PROGRAM TELNET_PRINT_DEMO_1
VAR
	COUNT_BR_1: COUNT_BR;
	READY: BOOL;
	TON_1: TON;
	TEXT: STRING;
	TEXT_ATTRIBUTE: BYTE;
	GEN_SIN_1: GEN_SIN;
	X_POS: BYTE;
	Y_POS: BYTE;
	GEN_SIN_2: GEN_SIN;
	TELNET_PRINT: TELNET_PRINT;
	DONE: BOOL;
	IP_C: IP_C;
	S_BUF: NETWORK_BUFFER;
	IP_CONTROL: IP_CONTROL;
	R_BUF: NETWORK_BUFFER;
END_VAR
VAR // added by the converter: edge detectors and wires of the graphical bodies
    _w1, _w2 : ANY;
END_VAR

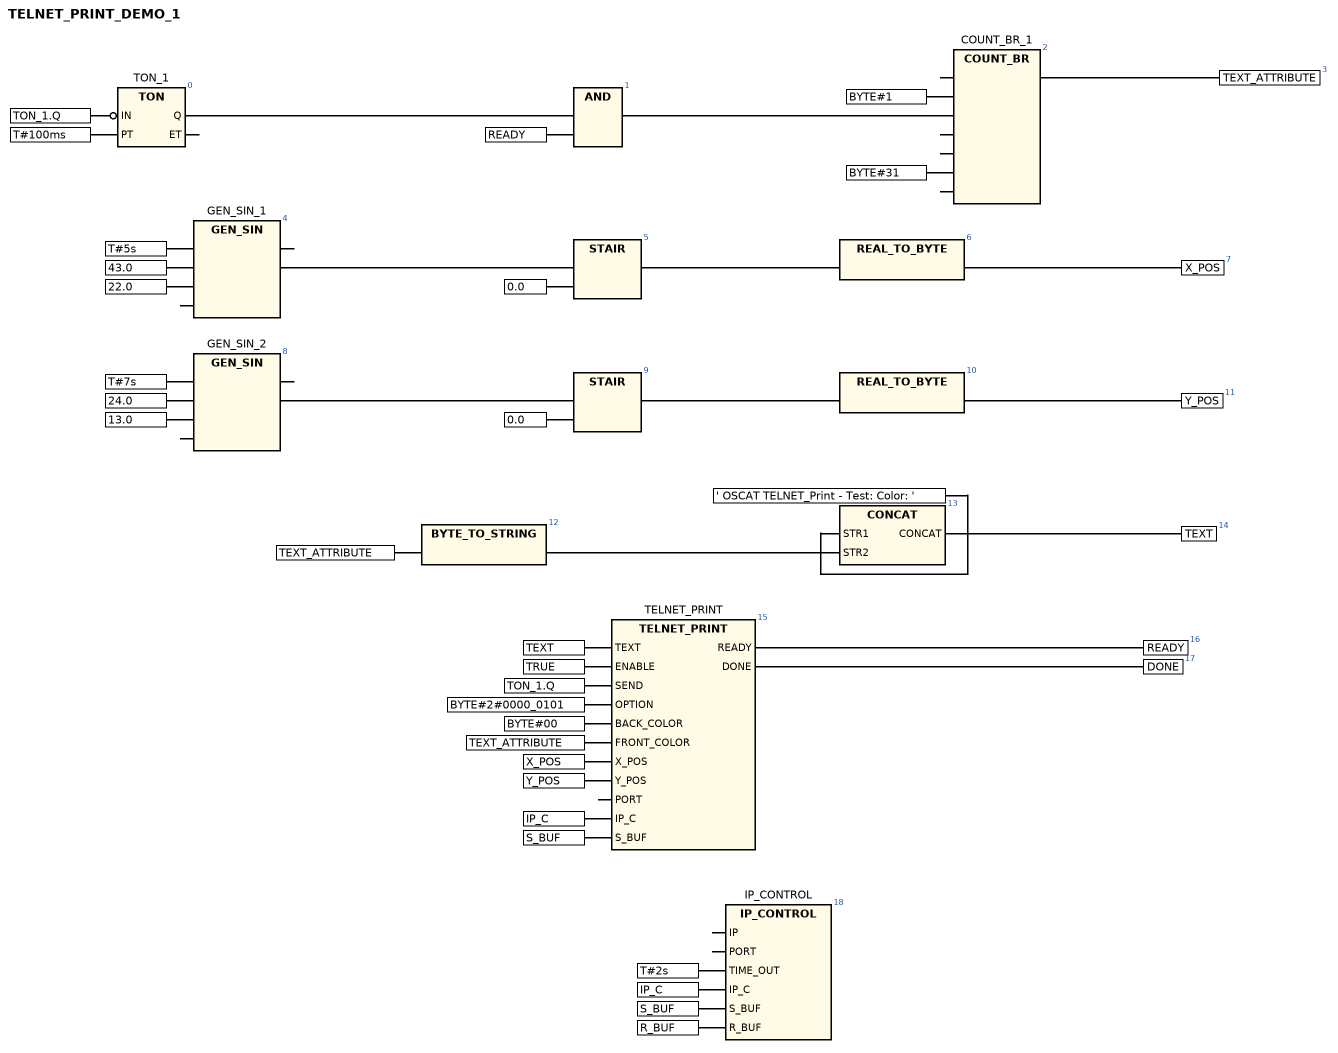
TON_1(IN := NOT TON_1.Q, PT := T#100ms); // TON
COUNT_BR_1(_in2 := BYTE#1, _in3 := TON_1.Q AND READY, _in6 := BYTE#31); // COUNT_BR
TEXT_ATTRIBUTE := COUNT_BR_1._out1;
GEN_SIN_1(_in1 := T#5s, _in2 := 43.0, _in3 := 22.0); // GEN_SIN
_w1 := STAIR(GEN_SIN_1._out2, 0.0);
X_POS := REAL_TO_BYTE(_w1);
GEN_SIN_2(_in1 := T#7s, _in2 := 24.0, _in3 := 13.0); // GEN_SIN
_w2 := STAIR(GEN_SIN_2._out2, 0.0);
Y_POS := REAL_TO_BYTE(_w2);
TEXT := CONCAT(STR1 := ' OSCAT TELNET_Print - Test: Color: ', STR2 := BYTE_TO_STRING(TEXT_ATTRIBUTE));
TELNET_PRINT(
    TEXT := TEXT,
    ENABLE := TRUE,
    SEND := TON_1.Q,
    OPTION := BYTE#2#0000_0101,
    BACK_COLOR := BYTE#00,
    FRONT_COLOR := TEXT_ATTRIBUTE,
    X_POS := X_POS,
    Y_POS := Y_POS,
    IP_C := IP_C,
    S_BUF := S_BUF);
READY := TELNET_PRINT.READY;
DONE := TELNET_PRINT.DONE;
IP_CONTROL(TIME_OUT := T#2s, IP_C := IP_C, S_BUF := S_BUF, R_BUF := R_BUF);

END_PROGRAM

(* stored: Version 1.1.0.1, ProductVersion 3.1.4024.0
   POU TELNET_PRINT_DEMO_1: Id {2e5de67a-0134-4b82-b02c-8b78f5d584ed}, SpecialFunc None *)
